(* PLC project CHL-DZ-BJDX-11 宁波数字孪生（东方理工）研究院制备薄层色谱全自动化工作站.project, Inovance company InoProShop(V1.9.1.6) InoProShop(V1.9.1.6) *)
(* stored: creationDateTime 2026-06-20T14:17:56.4556244, modificationDateTime 2026-06-18T22:35:27.3049867 *)

TYPE HMI_Servo : STRUCT
  position : ARRAY[1..10] OF LREAL;
  write : ARRAY[1..10] OF BOOL;
  execute : ARRAY[1..10] OF BOOL;
END_STRUCT;
END_TYPE

TYPE servo : STRUCT
  xHome : BOOL;  (* 回原点命令 *)
  xJogPos : BOOL;  (* 正方向点动 *)
  xJogNeg : BOOL;  (* 负方向点动 *)
  xStop : BOOL;  (* 停止命令 *)
  xMoveAbs : BOOL;  (* 绝对运动启动 *)
  xMoveRel : BOOL;  (* 相对运动启动 *)
  XReset : BOOL;  (* 轴复位 *)
  fAbsTarget : LREAL;  (* 绝对位置目标 *)
  fRelTarget : LREAL;  (* 相对运动距离 *)
  fVelocity : LREAL;  (* 运行速度 *)
  fAcc : LREAL;  (* 加速度 *)
  fDec : LREAL;  (* 减速度 *)
  fJogVel : LREAL;  (* 点动速度 *)
  bEnabled : BOOL;  (* 轴使能状态 *)
  bHomed : BOOL;  (* 原点完成 *)
  bBusy : BOOL;  (* 轴忙状态 *)
  bError : BOOL;  (* 轴报警 *)
  iErrorCode : DINT;  (* 错误代码 *)
  fActPos : LREAL;  (* 实际位置 *)
  fActVel : LREAL;  (* 实际速度 *)
  bAbMoveDone : BOOL;  (* 绝对运动完成 *)
  bReMoveDone : BOOL;  (* 相对运动完成 *)
END_STRUCT;
END_TYPE

{attribute 'qualified_only'}
{attribute 'strict'}
TYPE EN_功能块状态 : (停止 := 0, 运行 := 1, 故障 := 2, 急停 := 3, 初始化 := 4);
END_TYPE
